FUNCTION_BLOCK ToFinalTreatment_HMI (* Service Interface Function Block Type *)
  (* Standard: 61499-2 *)
  (* Version 0.0, 6/21/2026, Schneider Electric, template *)
  PACKAGE SE.Nereda;
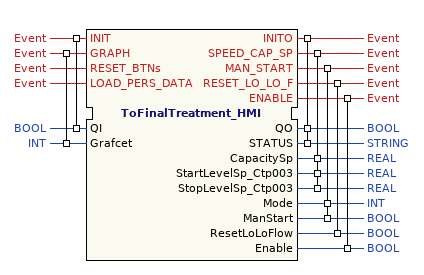
  EVENT_INPUT
    INIT WITH QI;
    GRAPH WITH Grafcet;
    RESET_BTNs;
    LOAD_PERS_DATA;
  END_EVENT
  EVENT_OUTPUT
    INITO WITH QO, STATUS;
    SPEED_CAP_SP WITH CapacitySp, StartLevelSp_Ctp003, StopLevelSp_Ctp003;
    MAN_START WITH ManStart, Mode;
    RESET_LO_LO_F WITH ResetLoLoFlow;
    ENABLE WITH Enable;
  END_EVENT
  VAR_INPUT
    QI : BOOL;
    Grafcet : INT;
  END_VAR
  VAR_OUTPUT
    QO : BOOL; (* Event Output Qualifier *)
    STATUS : STRING; (* Service Status *)
    CapacitySp : REAL;
    StartLevelSp_Ctp003 : REAL;
    StopLevelSp_Ctp003 : REAL;
    Mode : INT;
    ManStart : BOOL;
    ResetLoLoFlow : BOOL;
    Enable : BOOL;
  END_VAR
  SERVICE /
    SEQUENCE 
    END_SEQUENCE
  END_SERVICE
END_FUNCTION_BLOCK
